{attribute 'GeneratedUsingTerminal: EL6692-0002-0016'}
{attribute addProperty BoxType "EL6692-0002-0016"}
{attribute addProperty Id "EtcSlaveTerminalBaseSYNC_InputsAT %I*SYNC_Inputs_462ED3216IO_InputsEMPTY_STRUCTURE0IO_OutputsEMPTY_STRUCTURE0WcStateAT %I*WcState_9091E0EB2InfoDataAT %I*InfoData_90184F0C16"}
{attribute addProperty CRC "1319115998"}
{attribute addProperty Size "24"}
TYPE EL6692_4EA01CDE EXTENDS EtcSlaveTerminalBase :
STRUCT
	{attribute addProperty Name "SYNC_Inputs"}
	SYNC_Inputs : SYNC_Inputs_462ED321;
	{attribute addProperty Name "IO_Inputs"}
	IO_Inputs : EMPTY_STRUCTURE;
	{attribute addProperty Name "IO_Outputs"}
	IO_Outputs : EMPTY_STRUCTURE;
	{attribute addProperty Name "WcState"}
	WcState : WcState_9091E0EB;
	{attribute addProperty Name "InfoData"}
	InfoData : InfoData_90184F0C;
END_STRUCT
END_TYPE

(* stored: Version 1.2.0.0, ProductVersion 3.1.4024.9
   DUT EL6692_4EA01CDE: Id {96891174-9918-4001-b177-0aa7255093d0} *)
